(* PLC project CoDeSys External Library Template, WAGO e!COCKPIT e!COCKPIT, author 3S - Smart Software Solutions GmbH *)
(* stored: creationDateTime 2019-10-29T12:37:19.3649087, version 3.5.5.30, modificationDateTime 2019-10-29T12:36:39.3744516, organization 3S - Smart Software Solutions GmbH *)
(* Library project template with all possible element types, docu and a sample project structure *)

(* values of enumPPPSFriskoATTOM1STrybPracy: Zima: Zima; Lato: Lato; Auto: Automatyczny - przełączenie trybów uzależnione od temperatury zewnętrznej *)

(* Autor: Artur Wyszomirski, 22.05.2019 Prawa majątkowe: Solwena Sp. z o.o., Aktualizacje: Opis: enum służy do obsługi Trybów pracy fb węzła Frisko ATTO M1S na budynkach PPP Sopot (ENGIE) *)
{attribute 'qualified_only'}
{attribute 'strict'}
TYPE enumPPPSFriskoATTOM1STrybPracy : (Zima := 0, Lato := 1, Auto := 2);
END_TYPE
